// SIMATIC S7-200 SMART project (STEP 7-Micro/WIN SMART), CPU ST20

ORGANIZATION_BLOCK MAIN:OB1
TITLE=Program Comments
BEGIN
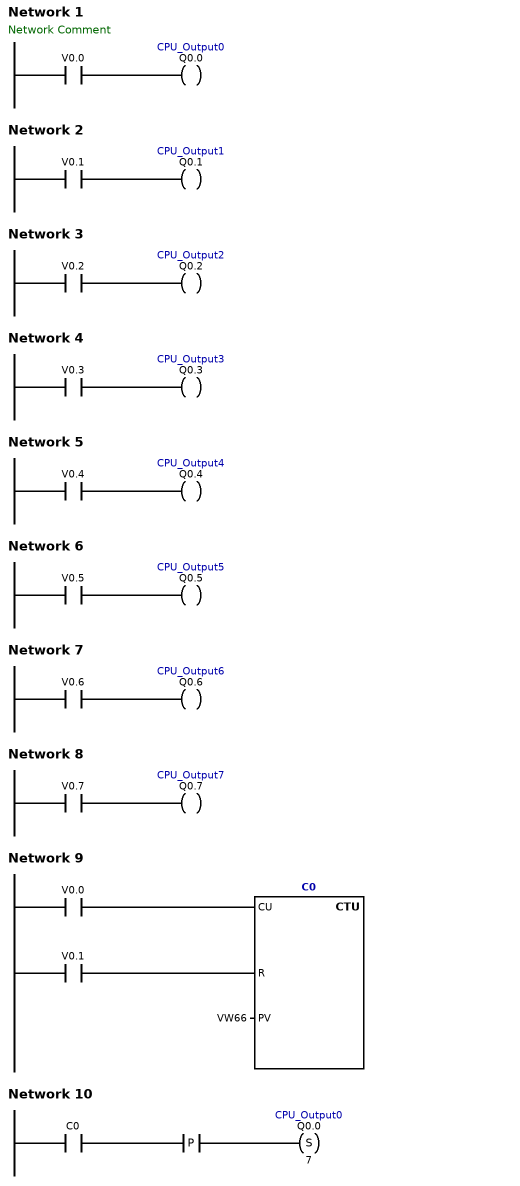
Network 1
// Network Comment
LD     V0.0
=      CPU_Output0:Q0.0
Network 2
LD     V0.1
=      CPU_Output1:Q0.1
Network 3
LD     V0.2
=      CPU_Output2:Q0.2
Network 4
LD     V0.3
=      CPU_Output3:Q0.3
Network 5
LD     V0.4
=      CPU_Output4:Q0.4
Network 6
LD     V0.5
=      CPU_Output5:Q0.5
Network 7
LD     V0.6
=      CPU_Output6:Q0.6
Network 8
LD     V0.7
=      CPU_Output7:Q0.7
Network 9
LD     V0.0
LD     V0.1
CTU    C0, VW66
Network 10
LD     C0
EU
S      CPU_Output0:Q0.0, 7
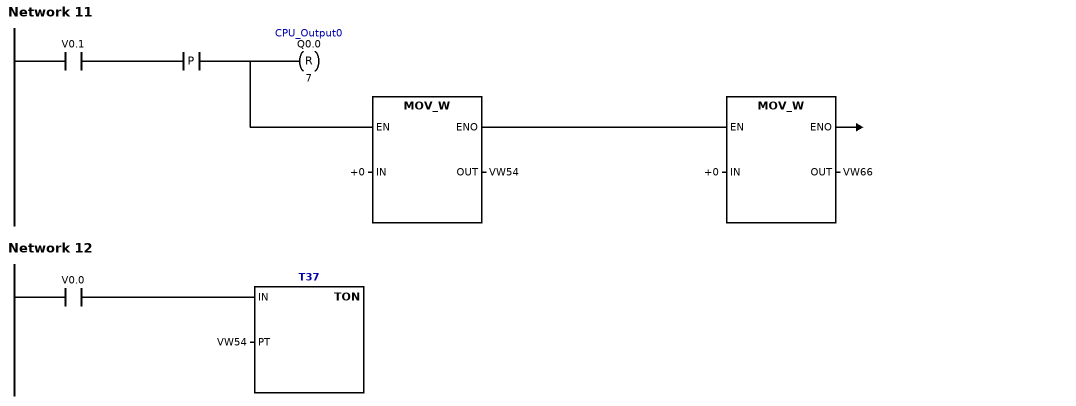
Network 11
LD     V0.1
EU
R      CPU_Output0:Q0.0, 7
MOVW   +0, VW54
AENO
MOVW   +0, VW66
Network 12
LD     V0.0
TON    T37, VW54
END_ORGANIZATION_BLOCK
